INTERFACE I_AliasDatatype EXTENDS I_UserDefinedDatatype

PROPERTY PUBLIC BaseDatatype : I_Datatype
GET
END_GET
END_PROPERTY

END_INTERFACE

(* stored: Version 1.1.0.1, ProductVersion 3.1.4024.12
   Itf I_AliasDatatype: Id {98310e30-586c-0f89-22af-eef9ccde9ada}
   Property BaseDatatype: Id {2c389239-8a6a-04a5-18f5-d35df619501e}
   Get Get: Id {fadc50f7-b906-04c6-19a3-10cc8bf79356} *)
